FUNCTION_BLOCK "GCS7_E_MessageCtrl"	// FB 25
TITLE = MSG
//  
//COPYRIGHT:    (C) 1996 BY  BUHLER LTD.
//                           CH-9240 UZWIL  SWITZERLAND
//
//PRODUCT:      GCS7
//
//TITLE:        ELEMENT Control Message
//
//-------------------------------------------------------------------------
//
//IDENT:        AUTHOR:             DEPT:                       DATE:
//
//FB25.2.0      A. Egli             CT3                        17-Jun-2002
//              New Release with one block 
//FB25.1A       A.Egli              AEE61                      05-Feb-1997
//              1st Release in S7
//
//-------------------------------------------------------------------------
//
//PURPOSE:      MANUAL : see [MSGxxMAN]
//              Can send up to 16 diverent message to host
//
//RESTRICTIONS: S7
//              ACCU2: Pointer to dynamic datas of the element
//              ACCU1: Pointer to parameter datas of the element
//
//-------------------------------------------------------------------------
//
//=======================================================
//Log Message: 
//------------------------------------------------------
//0    Inp0           
//1    Inp1         
//     :  
//     :  
//14   Inp14      
//15   Inp15      
//
//=======================================================
//StCode:  State               
//------------------------------------------------------
//0    Inp0           
//1    Inp1         
//     :  
//     :  
//14   Inp14      
//15   Inp15      
//16   OK     
//
//
AUTHOR : EA
FAMILY : GCS7LL
NAME : MSG
VERSION : 2.0
VAR
  StCode : INT ;	//Element state code
  InMsg0 : BOOL ;	//Send Message 0
  InMsg1 : BOOL ;	//Send Message 1
  InMsg2 : BOOL ;	//Send Message 2
  InMsg3 : BOOL ;	//Send Message 3
  InMsg4 : BOOL ;	//Send Message 4
  InMsg5 : BOOL ;	//Send Message 5
  InMsg6 : BOOL ;	//Send Message 6
  InMsg7 : BOOL ;	//Send Message 7
  InMsg8 : BOOL ;	//Send Message 8
  InMsg9 : BOOL ;	//Send Message 9
  InMsg10 : BOOL ;	//Send Message 10
  InMsg11 : BOOL ;	//Send Message 11
  InMsg12 : BOOL ;	//Send Message 12
  InMsg13 : BOOL ;	//Send Message 13
  InMsg14 : BOOL ;	//Send Message 14
  InMsg15 : BOOL ;	//Send Message 15
  OutFlag0 : BOOL ;	//Message 0 done
  OutFlag1 : BOOL ;	//Message 1 done
  OutFlag2 : BOOL ;	//Message 2 done
  OutFlag3 : BOOL ;	//Message 3 done
  OutFlag4 : BOOL ;	//Message 4 done
  OutFlag5 : BOOL ;	//Message 5 done
  OutFlag6 : BOOL ;	//Message 6 done
  OutFlag7 : BOOL ;	//Message 7 done
  OutFlag8 : BOOL ;	//Message 8 done
  OutFlag9 : BOOL ;	//Message 9 done
  OutFlag10 : BOOL ;	//Message 10 done
  OutFlag11 : BOOL ;	//Message 11 done
  OutFlag12 : BOOL ;	//Message 12 done
  OutFlag13 : BOOL ;	//Message 13 done
  OutFlag14 : BOOL ;	//Message 14 done
  OutFlag15 : BOOL ;	//Message 15 done
  Par : STRUCT
   ParObjectNo : INT ;	//Is used for communication with PC, e.g. for message
   ParMsgType : INT ;	//Is used for message (translation of state)
   ParHornCode : INT ;	//Is used by horn module
   ParDisable : STRUCT 	//Disable Message
    Msg0 : BOOL ;
    Msg1 : BOOL ;
    Msg2 : BOOL ;
    Msg3 : BOOL ;
    Msg4 : BOOL ;
    Msg5 : BOOL ;
    Msg6 : BOOL ;
    Msg7 : BOOL ;
    Msg8 : BOOL ;
    Msg9 : BOOL ;
    Msg10 : BOOL ;
    Msg11 : BOOL ;
    Msg12 : BOOL ;
    Msg13 : BOOL ;
    Msg14 : BOOL ;
    Msg15 : BOOL ;
   END_STRUCT ;
   ParHornOff : STRUCT 	//Disable Horn
    Msg0 : BOOL ;
    Msg1 : BOOL ;
    Msg2 : BOOL ;
    Msg3 : BOOL ;
    Msg4 : BOOL ;
    Msg5 : BOOL ;
    Msg6 : BOOL ;
    Msg7 : BOOL ;
    Msg8 : BOOL ;
    Msg9 : BOOL ;
    Msg10 : BOOL ;
    Msg11 : BOOL ;
    Msg12 : BOOL ;
    Msg13 : BOOL ;
    Msg14 : BOOL ;
    Msg15 : BOOL ;
   END_STRUCT ;
  END_STRUCT ;
END_VAR
VAR_TEMP
  tmpLOGvalue : WORD ;	//LOG value
  tmpReport : BOOL ;	//Global LOG all
  tmpOffsetInstanzDB : DINT ;
  tmpLenDyn : DINT ;
  tmpCntBit : DINT ;
  tmpAddrDynLoop : DINT ;
  tmpAddrParDisable : DINT ;
END_VAR
BEGIN
NETWORK
TITLE =  Start Global
      L     16;
      T     #tmpLenDyn;	//--> Len dynamic data in byte
      TAR2;
      L     DW#16#FFFFFF;
      AD;
      L     P##Par;
      +D;
      L     P#6.0;	//P##ParDisable
      +D;
      T     #tmpAddrParDisable;
NETWORK
TITLE = PC Control
//=== Test Object number =====================
      L     "SYS_DirectCtrlDB".PC.ObjectNo;	//PCControl.ObjectNo
      L     #Par.ParObjectNo;	//Input ObjectNo
      <>I;
      JC    Ctrl;
//=== Test OType      ========================
      L     1025;	//Input object type
      L     "SYS_DirectCtrlDB".PC.ObjectType;	//PCControl.ObjectType
      <>I;
      JC    Ctrl;
//=== Test Handshake =========================
      A     "SYS_DirectCtrlDB".PC.Hsk.FExamine;	// Handshake.FExamine
      JC    pExa;
      L     2;	// FcInit
      UC    "SYS_DirectCtrl";
      JU    Ctrl;
// Write parameter 
// Write new commands from PC to Interface of group 
// Examine
pExa: TAR2;	// Address Dynamic datas
      T     "SYS_DirectCtrlDB".GC.InDynAddr;	// -->PCControl.GC.InDynAddr
      L     #tmpLenDyn;	// Length Dynamic datas
      T     "SYS_DirectCtrlDB".GC.InDynLen;	// -->PCControl.GC.InDynLen
      L     0;
      T     "SYS_DirectCtrlDB".GC.InParaAddr;	// -->PCControl.GC.InParaAddr
      T     "SYS_DirectCtrlDB".GC.InParaLen;	// -->PCControl.GC.InParaLen
      L     1;	// Code FcExamine
      UC    "SYS_DirectCtrl";
      L     10;	//Revision
      T     "SYS_DirectCtrlDB".GC.Revision;
NETWORK
TITLE = AllState
NETWORK
TITLE = Log
//Message Type: 0 to 15 
//O = InMsg0
//15= InMsg15
// 
// Init Flag msg done (OutFlagXx) if InMsgXx=0
Ctrl: L     DIW [AR2,P#2.0];	// Load  Bit pattern InMsg0 ...InMsg15
      L     DIW [AR2,P#4.0];	// Load  Bit pattern OutFlag0 ...OutFlag15
      AW;
      T     DIW [AR2,P#4.0];	// Reset Bits pattern OutFlag0 ...OutFlag15
// 
// Test new Message to send;
      TAR2  #tmpAddrDynLoop;
      L     16;
NEX1: T     #tmpCntBit;
      LAR1  #tmpAddrParDisable;
      AN    DIX [AR1,P#0.0];	// ParDisable.MsgXx
      LAR1  #tmpAddrDynLoop;
      A     DIX [AR1,P#2.0];	// InMsgXx
      AN    DIX [AR1,P#4.0];	// OutFlagXx
      S     DIX [AR1,P#4.0];	// OutFlagXx
      JC    LOG;
      +AR1  P#0.1;
      TAR1  #tmpAddrDynLoop;
      L     #tmpAddrParDisable;
      L     P#0.1;
      +D;
      T     #tmpAddrParDisable;
      L     #tmpCntBit;
      LOOP  NEX1;
      JU    OUT;
LOG:  L     B#(4, 16);	//MessageClass Info ""Message 16"
      L     #tmpCntBit;
      -I;
      T     #tmpLOGvalue;
      LAR1  #tmpAddrParDisable;
      A     DIX [AR1,P#2.0];	// ParHornOff.MsgXx
      JC    Log3;
      CALL  "SYS_Horn_Code" (
           FcCode                   := 1,
           ParObjectType            := 1025,
           ParObjectNo              := #Par.ParObjectNo,
           ParHornCode              := #Par.ParHornCode);
Log3: CALL  "GCS7_LogConvert" (
           ObjectNo                 := #Par.ParObjectNo,
           MsgType                  := #Par.ParMsgType,
           ClassMsgTxt              := #tmpLOGvalue,
           OType                    := 1025);	// LOG Message Converter / Entry / Contains Class and TextNo
NETWORK
TITLE = State Code
OUT:  LAR1  AR2;
      L     16;
NEX2: T     #tmpCntBit;
      A     DIX [AR1,P#2.0];	// InMsgXx
      JC    STC;
      +AR1  P#0.1;
      L     #tmpCntBit;
      LOOP  NEX2;
      L     16;
      JU    OK;
STC:  L     16;
      L     #tmpCntBit;
      -I;	// Code: fault
OK:   L     #StCode;	// Old state code
      TAK;
      T     #StCode;	// Save state code
      <>I;
      L     3;	// Load code for CBit methode
      CC    "SYS_CBitCtrl";
END_FUNCTION_BLOCK

FUNCTION_BLOCK "GCS7_E_DFCO"	// FB 26
TITLE = DFCO
//  
//COPYRIGHT:    (C) 1996  BUHLER AG, CH-9240 UZWIL, SWITZERLAND
//
//PRODUCT:      GCS7
//
//TITLE:        Element Control DFCO
//              (GCPROVB Revision 11)  
//
//-------------------------------------------------------------------------
//
//IDENT:        AUTHOR:             DEPT:                       DATE:
//
//FB26.2.3      A. Egli             BASE                        20-Okt-2008
//              For timeout starting check ParDFCO_Only
//FB26.2.2      A.Egli              CT3                         26-Sep-2007
//              Do not set "GCS7_Gr_InHeavyStartup" if ParDFCO_Only=1         
//FB26.2.1      A.Egli              CT3                         11-Sep-2007
//              Send Log Message if Alarmnumber changes from 0->X          
//FB26.2.0      A.Egli              CT3                         14-Feb-2007
//              New Tag names           
//FB26.1.4      B.Thoma             FU591                       02-Dez-2006
//              Delete all actual values as long Profibus fault           
//FB26.1.3      B.Thoma             FU91                        28-Nov-2006
//              Invert HL DFAV ; StCode Fan           
//FB26.1.2      B.Thoma             FU92                        18-Apr-2006
//              Flapbox changed 
//              FeedRoll State changed            
//FB26.1.1      A.Egli              CT3                         01-Dec-2005
//              Parameter Upload Change DBD86-->DBD88
//FB26.1.0      A.Egli              CT3                         06-Oct-2005
//              1st Release in S7
//
//-------------------------------------------------------------------------
//
//PURPOSE:      MANUAL : see [DFCOxxMAN]
//
//RESTRICTIONS: S7
//             
//=======================================================
//Log Message: 
//------------------------------------------------------
//0     = Fault Cancelled
//1..89 = AlarmLC : Alarmnumber see manual of MEAF
//90    = Fault Remote Control
//91    = StStopped
//92    = StStarted
//95    = WrongValue
//96    = Communication fault
//97    = 
//98    = 
//99    = Collected alarm
//
//=======================================================
//StCode:  State               
//------------------------------------------------------
// StFault                 32
// StStopped                1
// StStarting               2
// StStarted.Wait           3
// StStarted.Feeding        4
// StStopping               7
// StWarning                8
//
AUTHOR : EA
FAMILY : GCS7LL
NAME : DFCO
VERSION : 2.3
VAR
  StCode : INT ;	// State as code 32=StFault 1=StStopped 2=StStarting 3=StStartedWait 4=StStartedF
  spare20 : BOOL ;
  spare21 : BOOL ;
  spare22 : BOOL ;
  InReqStartRev : BOOL ;	//Mill must start reverse
  InReqStartFwd : BOOL ;	//Mill must start forward
  spare25 : BOOL ;	//1=Activate automatic control mode (CTRL.MODE)
  InHeavyFractionOpen : BOOL ;
  spare27 : BOOL ;
  spare30 : BOOL ;
  spare31 : BOOL ;	//
  CmdNext : BOOL ;	// Pulse to start the next motor in automatic mode
  CmdFaultReset : BOOL ;	// Command to reset fault
  InLocal : BOOL ;	// Local mode, accept all faults
  InManual : BOOL ;	//
  InReport : BOOL ;	//
  spare37 : BOOL ;
  InHWStop : BOOL ;	//HW stop is detected, no fault
  InDPFault : BOOL ;	//DP-Fault is detected, no fault
  InSimulation : BOOL ;	//Simulation with DPSim
  OutComFault : BOOL ;	//Communication fault
  OutStartwarning : BOOL ;	//Not used
  spare45 : BOOL ;
  spare46 : BOOL ;
  spare47 : BOOL ;
  StStopped : BOOL ;	//All motors are stopped
  StStarting : BOOL ;	//Not all relevant motors are started
  StStarted : BOOL ;	//All used motors are started
  StStopping : BOOL ;	//Any motor is stopping
  StFault : BOOL ;	//Any relevant element has a fault
  spare0505 : BOOL ;	//
  spare0506 : BOOL ;	//
  spare0507 : BOOL ;	//
  Mill1 : STRUCT
   InEnable : BOOL ;	//Automatic Mode
   InUsed : BOOL ;	//Automatic Mode
   InEnableFeed : BOOL ;	//Automatic Mode
   InBrake : BOOL ;	//Automatic Mode: Stop with break
   InFast : BOOL ;	//Run motor with fast speed
   spare05 : BOOL ;
   spare06 : BOOL ;
   spare07 : BOOL ;
   CmdOff : BOOL ;	//Manual Mode
   CmdOn : BOOL ;	//Manual Mode
   CmdFeedOff : BOOL ;	//Manual Mode
   CmdFeedOn : BOOL ;	//Manual Mode
   CmdBrake : BOOL ;	//Manual Mode
   spare15 : BOOL ;
   spare16 : BOOL ;
   InpFanStart : BOOL ;	//Fan is started
   OutpMotorFwd : BOOL ;	//Output run motor forward
   OutpMotorFast : BOOL ;	//Output run motor fast
   OutpMotorRev : BOOL ;	//Output run motor reverse
   OutpBrake : BOOL ;	//Output brake
   OutpFanStart : BOOL ;	//Output run fan
   OutLoaded : BOOL ;	//Read from DFCO
   OutWrongValue : BOOL ;
   OutScreenChangeReq : BOOL ;	//Srceen change is requested
   VarEdgeStarted : BOOL ;
   VarEdgeFault : BOOL ;
   Tar : STRUCT 	//Telegram Dataset 128
    InSetPoint : INT ;	//[%] Load control
    InScreen : INT ;	//[0.1mm] Sreen size
    spare1 : INT ;
    spare2 : INT ;
    spare3 : INT ;
    spare4 : INT ;
    EmptyTime : INT ;	//[0.1s]
    spare5 : INT ;
   END_STRUCT ;
   Act : STRUCT 	//Telegram Dataset 1
    OutLoadAct : INT ;	//[%]
    OutCurrentLoad : INT ;	//[0.1A]
    OutActPosSlide : INT ;	//[%]
    OutActTemperature : INT ;	//[0.1°C]
    OutStatusFlapBox : INT ;
    OutStatusMillMotor : INT ;
    spare1 : INT ;
    OutEmptyTime : INT ;	//[0.1s]
    spare2 : INT ;
    OutAlarmNo : INT ;
   END_STRUCT ;
   Motor : STRUCT
    StStopped : BOOL ;
    StStarting : BOOL ;
    StStartedFwd : BOOL ;
    StStopping : BOOL ;
    StFault : BOOL ;
    StStartedRev : BOOL ;
    StBrake : BOOL ;
   END_STRUCT ;
   OutScreenAct : INT ;	//[0.1mm] Actual screen
   spare1 : INT ;
   spare2 : INT ;
   spare3 : INT ;
   spare4 : INT ;
   spare5 : INT ;
   spare6 : INT ;
   Motor_StCode : INT ;	//StCode same as EL_Motor
   Vibration_StCode : INT ;	//StCode same as EL_DIC
   Automatic_StCode : INT ;	//StCode same as EL_DIC
   StandStill_StCode : INT ;	//StCode same as EL_DIC
   SwitchPanel_StCode : INT ;	//StCode same as EL_DIC
   EmergencyStop_StCode : INT ;	//StCode same as EL_DIC
   HLCone_StCode : INT ;	//StCode same as EL_DIC
   OutTimeStartedFwd : DINT ;	//[s] Not errasable time "Started"
   OutTimeStartedRev : DINT ;	//[s] Not errasable time "Started"
   OutTimeFaulted : DINT ;	//[s] Not errasable time "Faulted"
   OutCntStartup : DINT ;	//Not errasable counter of startup
   OutCntFault : DINT ;	//Not errasable counter of faults
  END_STRUCT ;
  Mill2 : STRUCT
   InEnable : BOOL ;	//Automatic Mode
   InUsed : BOOL ;	//Automatic Mode
   InEnableFeed : BOOL ;	//Automatic Mode
   InBrake : BOOL ;	//Automatic Mode: Stop with break
   InFast : BOOL ;	//Run motor with fast speed
   spare05 : BOOL ;
   spare06 : BOOL ;
   spare07 : BOOL ;
   CmdOff : BOOL ;	//Manual Mode
   CmdOn : BOOL ;	//Manual Mode
   CmdFeedOff : BOOL ;	//Manual Mode
   CmdFeedOn : BOOL ;	//Manual Mode
   CmdBrake : BOOL ;	//Manual Mode
   spare15 : BOOL ;
   spare16 : BOOL ;
   InpFanStart : BOOL ;	//Fan is started
   OutpMotorFwd : BOOL ;	//Output run motor forward
   OutpMotorFast : BOOL ;	//Output run motor fast
   OutpMotorRev : BOOL ;	//Output run motor reverse
   OutpBrake : BOOL ;	//Output brake
   OutpFanStart : BOOL ;	//Output run fan
   OutLoaded : BOOL ;	//Read from DFCO
   OutWrongValue : BOOL ;
   OutScreenChangeReq : BOOL ;	//Srceen change is requested
   VarEdgeStarted : BOOL ;
   VarEdgeFault : BOOL ;
   Tar : STRUCT 	//Telegram Dataset 128
    InSetPoint : INT ;	//[%] Load control
    InScreen : INT ;	//[0.1mm] Sreen size
    spare1 : INT ;
    spare2 : INT ;
    spare3 : INT ;
    spare4 : INT ;
    EmptyTime : INT ;	//[0.1s]
    spare5 : INT ;
   END_STRUCT ;
   Act : STRUCT 	//Telegram Dataset 1
    OutLoadAct : INT ;	//[%]
    OutCurrentLoad : INT ;	//[0.1A]
    OutActPosSlide : INT ;	//[%]
    OutActTemperature : INT ;	//[0.1°C]
    OutStatusFlapBox : INT ;
    OutStatusMillMotor : INT ;
    spare1 : INT ;
    OutEmptyTime : INT ;	//[0.1s]
    spare2 : INT ;
    OutAlarmNo : INT ;
   END_STRUCT ;
   Motor : STRUCT
    StStopped : BOOL ;
    StStarting : BOOL ;
    StStartedFwd : BOOL ;
    StStopping : BOOL ;
    StFault : BOOL ;
    StStartedRev : BOOL ;
    StBrake : BOOL ;
   END_STRUCT ;
   OutScreenAct : INT ;	//[0.1mm] Actual screen
   spare1 : INT ;
   spare2 : INT ;
   spare3 : INT ;
   spare4 : INT ;
   spare5 : INT ;
   spare6 : INT ;
   Motor_StCode : INT ;	//StCode same as EL_Motor
   Vibration_StCode : INT ;	//StCode same as EL_DIC
   Automatic_StCode : INT ;	//StCode same as EL_DIC
   StandStill_StCode : INT ;	//StCode same as EL_DIC
   SwitchPanel_StCode : INT ;	//StCode same as EL_DIC
   EmergencyStop_StCode : INT ;	//StCode same as EL_DIC
   HLCone_StCode : INT ;	//StCode same as EL_DIC
   OutTimeStartedFwd : DINT ;	//[s] Not errasable time "Started"
   OutTimeStartedRev : DINT ;	//[s] Not errasable time "Started"
   OutTimeFaulted : DINT ;	//[s] Not errasable time "Faulted"
   OutCntStartup : DINT ;	//Not errasable counter of startup
   OutCntFault : DINT ;	//Not errasable counter of faults
  END_STRUCT ;
  OutActFeedRoll : INT ;	//[Hz] Actual frequence feed roll
  spare208 : DINT ;	//StCode same as EL_DIC
  spare212 : DINT ;
  spare216 : DINT ;
  FlapBox : STRUCT
   StMill1 : BOOL ;
   StMiddle : BOOL ;
   StMill2 : BOOL ;
   StNoPosition : BOOL ;
  END_STRUCT ;
  FlapBox_StCode : INT ;	//StCode same as EL_VLS4
  FeedRoll_StCode : INT ;	//StCode same as EL_Motor
  Fan_StCode : INT ;	//StCode same as EL_Motor
  LL_FeedHopper_StCode : INT ;	//StCode same as EL_DIC
  HL_DFAV_StCode : INT ;	//StCode same as EL_DIC
  MagnetDoor_StCode : INT ;	//StCode same as EL_DIC
  HeavyParticalFlap_StCode : INT ;	//StCode same as EL_DIC
  spare118 : INT ;
  spare220 : DINT ;
  spare224 : DINT ;
  spare228 : DINT ;
  OutAlarmNoLog : INT ;	//Last textnumber send to log
  InpDFCO : STRUCT 	//WAGO/MEAF Inputs of DFCO
   I00_LL_FeedHopper : BOOL ;	//DFAV: Inlet level DFAV (1=covered)
   I01_HL_DFAV : BOOL ;	//DFAV: High level DFAV (1=Covered)
   I02_HeavyParticleFlap : BOOL ;	//DFAV: Heavy particle flap closed (1=end position)
   I03_MagnetDoorClosed : BOOL ;	//DFAV: Door interlocking heavy particle flap (1=closed)
   I04_LSFlapBox : BOOL ;	//DFAV: LS of middle position (1=dedected)
   I05 : BOOL ;
   I06 : BOOL ;
   I07_24VOk : BOOL ;	//DFAV: Fuse control of DFCO (1=ok)
   spare9 : BYTE ;
   I20_ButtonCone1 : BOOL ;	//DFZK Mill 1: Button open/close cone
   I21_ButtonHeavyFlap1 : BOOL ;	//DFZK Mill 1: Button open heavy particle flap
   I22_KeySwitchAuto1 : BOOL ;	//DFZK Mill 1: Key switch Automatic/Hand (1=Hand)
   I23_SwitchPanel1 : BOOL ;	//DFZK Mill 1: Connection box (1= inactive)
   I24_StandStill1 : BOOL ;	//DFZK Mill 1: Standstill (1=Standstill)
   I25_EmergencyStop1 : BOOL ;	//DFZK Mill 1: Cone interlocking (1=not interlocked)
   I26_EmergencySwitch1 : BOOL ;	//DFZK Mill 1: Emergency switch(1=ok)
   I27_HL_Cone1 : BOOL ;	//DFZK Mill 1: HL outlet cone (1=uncovered)
   spare11 : BYTE ;
   I40_ButtonCone2 : BOOL ;	//DFZK Mill 2: Button open/close cone
   I41_ButtonHeavyFlap2 : BOOL ;	//DFZK Mill 2: Button open heavy particle flap
   I42_KeySwitchAuto2 : BOOL ;	//DFZK Mill 2: Key switch Automatic/Hand (1=Hand)
   I43_SwitchPanel2 : BOOL ;	//DFZK Mill 2: Connection box (1= inactive)
   I44_StandStill2 : BOOL ;	//DFZK Mill 2: Standstill (1=Standstill)
   I45_EmergencyStop2 : BOOL ;	//DFZK Mill 2: Cone interlocking (1=not interlocked)
   I46_EmergencySwitch2 : BOOL ;	//DFZK Mill 2: Emergency switch(1=ok)
   I47_HL_Cone2 : BOOL ;	//DFZK Mill 2: HL outlet cone (1=uncovered)
   spare13 : BYTE ;
   I60_VibrationDetector1 : BOOL ;	//DFZK Mill 1: Vibration detector (1=OK)
   I61_VibrationDetector2 : BOOL ;	//DFZK Mill 2: Vibration detector (1=OK)
   spare15 : BYTE ;
   I80_Release1 : BOOL ;	//DFZK Mill 1: Release feeding (1=released)
   I81_Start1 : BOOL ;	//DFZK Mill 1: Release motor (1=released)
   I82_RotarySpeed1 : BOOL ;	//DFZK Mill 1: Fast/Slow speed of motor (2=fast)
   I83_AckFan : BOOL ;	//DFZK Mill 1: Fan is running
   I84 : BOOL ;
   I85 : BOOL ;
   I86 : BOOL ;
   I87 : BOOL ;
   I90_Release2 : BOOL ;	//DFZK Mill 2: Release feeding (1=released)
   I91_Start2 : BOOL ;	//DFZK Mill 2: Release motor (1=released)
   I92_Speed2 : BOOL ;	//DFZK Mill 2: Fast/Slow speed of motor (1=fast)
   I93_Break : BOOL ;	//DFZK Mill 1/2: Stop with break (1=with break)
   spare18 : BYTE ;
   spare19 : BYTE ;
   spare20 : BYTE ;
   DI1_spare : BOOL ;
   DI2_spare : BOOL ;
   DI3_spare : BOOL ;
   DI4_spare : BOOL ;
   DI5_SlideEndPos1 : BOOL ;	//DFZK Mill 1: Slide end position
   DI6_SlidePulse1 : BOOL ;	//DFZK Mill 1: Slide pulse signal
   DI7_SlideEndPos2 : BOOL ;	//DFZK Mill 2: Slide end position
   DI8_SlidePulse2 : BOOL ;	//DFZK Mill 2: Slide pulse signal
  END_STRUCT ;
  OutpDFCO : STRUCT 	//WAGO/MEAF Outpus of DFCO
   O00_HeavyParticleClose : BOOL ;	//DFAV: Heavy particle flap close
   O01_HeavyParticleOpen : BOOL ;	//DFAV: Heavy particle flap open
   O02_FlapCylinderExtend : BOOL ;	//DFAV: Flap box cylinder extend
   O03_FlapCylinderRetract : BOOL ;	//DFAV: Flap box cylinder retract
   spare9 : BYTE ;
   O20_LampAlarm1 : BOOL ;	//DFZK Mill 1: Lamp alarm (1=Alarm)
   O21_LampRelaseCone1 : BOOL ;	//DFZK Mill 1: Lamp cone adjustment
   O22_LampHeavyParticle : BOOL ;	//DFZK Mill 1: Lamp heavy particle flap
   spare11 : BYTE ;
   O40_LampAlarm2 : BOOL ;	//DFZK Mill 2: Lamp alarm (1=Alarm)
   O41_LampReleaseCone2 : BOOL ;	//DFZK Mill 2: Lamp cone adjustment
   O42_LampHeavyParticle : BOOL ;	//DFZK Mill 2: Lamp heavy particle flap
   O43 : BOOL ;
   O44 : BOOL ;
   O45 : BOOL ;
   O46 : BOOL ;
   O47 : BOOL ;
   O50_ConeOpen1 : BOOL ;	//DFZK Mill 1: Cone open
   O51_ConeClose1 : BOOL ;	//DFZK Mill 1: Cone close
   O52 : BOOL ;	//
   O53 : BOOL ;	//
   O54 : BOOL ;
   O55 : BOOL ;
   O56 : BOOL ;
   O57 : BOOL ;
   O60_ConeOpen2 : BOOL ;	//DFZK Mill 2: Cone open
   O61_ConeClose2 : BOOL ;	//DFZK Mill 2: Cone close
   spare15 : BYTE ;
   O80_Alarm1 : BOOL ;	//DFZK Mill 1: Alarm (1=no alarm)
   O81_StartMotor1 : BOOL ;	//DFZK Mill 1: Start motor forward
   O82_MotorFast1 : BOOL ;	//DFZK Mill 1: Start motor fast
   O83_MotorRev1 : BOOL ;	//DFZK Mill 1: Start motor reverse
   O84_Break1 : BOOL ;	//DFZK Mill 1: Brake motor
   O85_StartFan : BOOL ;	//DFZK Mill 1/2: Start fan
   O86 : BOOL ;
   O87 : BOOL ;
   O90_Alarm2 : BOOL ;	//DFZK Mill 2: Alarm (1=no alarm)
   O91_StartMotor2 : BOOL ;	//DFZK Mill 2: Start motor forward
   O92_MotorFast2 : BOOL ;	//DFZK Mill 2: Start motor fast
   O93_MotorRev2 : BOOL ;	//DFZK Mill 2: Start motor reverse
   O94_Break2 : BOOL ;	//DFZK Mill 2: Brake motor
   spare18 : BYTE ;
   spare19 : BYTE ;
   spare20 : BYTE ;
   DO1_SummaryAlarm : BOOL ;	//Summary alarm
   DO2 : BOOL ;
   DO3 : BOOL ;
   DO4_Slide1Open : BOOL ;	//Slide 1 open
   DO5_Slide1Close : BOOL ;	//Slide 1 close
   DO6_Slide2Open : BOOL ;	//Slide 2 open
   DO7_Slide2Close : BOOL ;	//Slide 2 close
   DO8 : BOOL ;
  END_STRUCT ;
  Command : STRUCT 	//Command for DFCO
   spare0 : BOOL ;	//1=Automatic/ 0=Manual
   AckStartRequest : BOOL ;	//Acknowledge Start Request
   ReqStartRev : BOOL ;	//Mill must start reverse
   ReqStartFwd : BOOL ;	//Mill must start forward
   HeavyFractionOpen : BOOL ;	//Heavy fraction flap is open
   ReqScreenChange1 : BOOL ;
   ReqScreenChange2 : BOOL ;
   AcceptNewDataReady : BOOL ;	//de: Quittierung neue Werte Bereit
   EnableMill1 : BOOL ;	//Enable to start mill 1
   MotorMill1Fast : BOOL ;
   UsedMill1 : BOOL ;
   BrakeMill1 : BOOL ;	//Stop mill 1
   EnableFeedMill1 : BOOL ;	//Enable Feed of mill 1
   AckFanStart : BOOL ;	//Fan is running
   spare16 : BOOL ;
   spare17 : BOOL ;
   EnableMill2 : BOOL ;	//Enable to start mill 1
   MotorMill2Fast : BOOL ;
   UsedMil12 : BOOL ;
   BrakeMill2 : BOOL ;	//Stop mill 1
   EnableFeedMill2 : BOOL ;	//Enable Feed of mill 1
   spare25 : BOOL ;
   spare26 : BOOL ;
   spare27 : BOOL ;
   CommandReady : BOOL ;	//de: Steuersignale gültig
   spare41 : BOOL ;
   spare42 : BOOL ;
   spare43 : BOOL ;
   spare44 : BOOL ;
   ResetAlarm : BOOL ;	//de: Alarm löschen
   NewSendData : BOOL ;	//de: Aenderung Sendedaten
   AcceptNewRcvData : BOOL ;	//de: Quittierung Aenderung Empfangsdatensatz
  END_STRUCT ;
  Status : STRUCT 	//Status from DFCO
   spare00 : BOOL ;
   ReqStartRequest : BOOL ;	//Start Request : DFCO like to start a motor
   Loaded1 : BOOL ;	//Mill 1 loaded with product
   Loaded2 : BOOL ;	//Mill 2 loaded with product
   spare04 : BOOL ;
   AckScreenChange1 : BOOL ;
   AckScreenChange2 : BOOL ;
   NewDataReady : BOOL ;	//de: Neue Werte Bereit
   O80Alarm1 : BOOL ;	//False=Alarm
   O81MotorFwd1 : BOOL ;	//Output run motor forward
   O82MotorFast1 : BOOL ;	//Output run motor fast
   O83MotorRev1 : BOOL ;	//Output run motor reverse
   O84Brake1 : BOOL ;	//Output brake
   O85FanStart : BOOL ;	//Output run fan
   spare16 : BOOL ;
   spare17 : BOOL ;
   O90Alarm2 : BOOL ;	//False=Alarm
   O91MotorFwd2 : BOOL ;	//Output run motor forward
   O92MotorFast2 : BOOL ;	//Output run motor fast
   O93MotorRev2 : BOOL ;	//Output run motor reverse
   O94Brake2 : BOOL ;	//Output brake
   spare25 : BOOL ;	//Output run fan
   spare26 : BOOL ;
   spare27 : BOOL ;
   spare30 : BOOL ;
   spare31 : BOOL ;
   spare32 : BOOL ;	//de: Stuerung Remote
   RemoteControlDP : BOOL ;	//de: Sollwertvorgabe Remote
   WrongValue : BOOL ;	//de: Falscher Sollwert
   SumFault : BOOL ;	//de: Sammelalarm
   AcceptNewSendData : BOOL ;	//de: Quittierung Aenderung Sendedaten
   NewRcvData : BOOL ;	//de: Aenderung Empfangsdaten
  END_STRUCT ;
  Par : STRUCT
   ParObjectNo : INT ;	//Is used for communication with PC, e.g. for message
   ParMsgType : INT ;	//Is used for message (translation of state)
   ParHornCode : INT ;	//Is used by horn module
   ParLogOff : BOOL ;	//Report is off
   ParManual : BOOL ;	//Manual mode without interlocking
   ParDFCO_Only : BOOL ;	//Only throughput regulation, no motors
   ParStartwarning : BOOL ;	//not used
   ParIOByteNo : INT ;	//PROFIBUS: Address of first input and output byte Profibus DP
   ParTimeOutStart : INT  := 50;	//[0.1s] After this time the motor must start
   OutTimeOutStart1 : INT ;	//[0.1s] Actual timeout time mill 1
   OutTimeOutStart2 : INT ;	//[0.1s] Actual timeout time mill 2
   Spare94 : DINT ;
   spare98 : DINT ;
   Spare94_1 : DINT ;
   HelpFlags : STRUCT 	//Aux. signal to retry fault message
    OutFaultResetDone : BOOL ;
    OutTestNewAlarm : BOOL ;
    OutFlagFaultResetDone : BOOL ;
    OutComFaultRead : BOOL ;
    OutComFaultSend : BOOL ;
   END_STRUCT ;
  END_STRUCT ;
END_VAR
VAR_TEMP
  tmpLOGvalue : WORD ;	//LOG value
  tmpReport : BOOL ;	//Global LOG all
  tmpFault : BOOL ;
  tmpLocal : BOOL ;
  tmpStarted : BOOL ;
  tmpStopped : BOOL ;
  tmpLenDyn : DINT ;
  tmpReturn : INT ;
  DPData : STRUCT
   StatusCommand : DWORD ;
   NrSndDataSet : BYTE ;	//de: Nummer Sendedatensatz
   IdxSndDataSet : BYTE ;	//de: Index Sendedatensatz
   NrRcvDataSet : BYTE ;	//de: Nummer Empfangsdatensatz
   IdxRcvDataSet : BYTE ;	//de: Index Empfangsdatensatz
   Data : ARRAY  [1 .. 4 ] OF DINT ;
  END_STRUCT ;
  Set1 : STRUCT
   OutLoadAct : INT ;	//[%]
   OutCurrentLoad : INT ;	//[0.1A]
   OutActPosSlide : INT ;	//[%]
   OutActTemperature : INT ;	//[0.1°C]
   OutStatusFlapBox : BYTE ;
   OutStatusMillMotor : BYTE ;
   OutActFeedFoll : BYTE ;	//[Hz] Actual frequence feed roll
   spare1 : BYTE ;
   OutEmptyTime : INT ;	//[0.1s]
   spare2 : BYTE ;
   OutAlarmNo : BYTE ;
  END_STRUCT ;
  tmpAddr : WORD ;
  tmpCnt : INT ;
  tmpRetVal : INT ;
  tmpBool : BOOL ;
END_VAR
BEGIN
NETWORK
TITLE =  Start Global
      L     298;
      T     #tmpLenDyn;	//--> Len dynamic data in byte
NETWORK
TITLE = PC Control
//=== Test Object number =====================
      L     "SYS_DirectCtrlDB".PC.ObjectNo;	//PCControl.ObjectNo
      L     #Par.ParObjectNo;	//Input ObjectNo
      <>I;
      JC    aEnd;
//=== Test OType  ========================
      L     1026;	//Input object type
      L     "SYS_DirectCtrlDB".PC.ObjectType;	//PCControl.ObjectType
      <>I;
      JC    aEnd;
//=== Test Handshake =========================
      A     "SYS_DirectCtrlDB".PC.Hsk.FExamine;	// Handshake.FExamine
      JC    aExa;
      A     "SYS_DirectCtrlDB".PC.Hsk.FDefineCmd;	// Handshake.FDefineCmd
      JC    aCmd;
      A     "SYS_DirectCtrlDB".PC.Hsk.FDefinePara;	// Handshake.FDefinePara
      JC    pPar;
aIni: L     2;	// FcInit
      UC    "SYS_DirectCtrl";
      JU    aEnd;
// Write parameter 
pPar: LAR1  P#DBX 58.0;
      L     P#6.0;
      +AR1;
// Write new commands from PC to Interface of group 
// Mill 1
aCmd: A     "SYS_DirectCtrlDB".PC.Cmd1[0];	//CmdBrakeMill1On
      AN    "GCS7_Gr_OutManualOff";	//Global.OutManualOff  [2.10]
      S     #Mill1.CmdBrake;
      A     "SYS_DirectCtrlDB".PC.Cmd1[1];	//CmdReqSlow
      R     #Command.MotorMill1Fast;
      A     "SYS_DirectCtrlDB".PC.Cmd1[2];	//CmdReqFast
      S     #Command.MotorMill1Fast;
      A     "SYS_DirectCtrlDB".PC.Cmd1[3];	//CmdReqRev
      S     #Command.ReqStartRev;
      R     #Command.ReqStartFwd;
      A     "SYS_DirectCtrlDB".PC.Cmd1[4];	//CmdReqFwd
      R     #Command.ReqStartRev;
      S     #Command.ReqStartFwd;
      A     "SYS_DirectCtrlDB".PC.Cmd1[8];	// CmdOff
      AN    "GCS7_Gr_OutManualOff";	//Global.OutManualOff  [2.10]
      S     #Mill1.CmdOff;
      A     "SYS_DirectCtrlDB".PC.Cmd1[9];	// CmdOn
      AN    "GCS7_Gr_OutManualOff";	//Global.OutManualOff  [2.10]
      S     #Mill1.CmdOn;
      A     "SYS_DirectCtrlDB".PC.Cmd1[6];	// CmdFeedOff
      AN    "GCS7_Gr_OutManualOff";	//Global.OutManualOff  [2.10]
      S     #Mill1.CmdFeedOff;
      A     "SYS_DirectCtrlDB".PC.Cmd1[7];	// CmdFeedOn
      AN    "GCS7_Gr_OutManualOff";	//Global.OutManualOff  [2.10]
      S     #Mill1.CmdFeedOn;
// Mill 2
      A     "SYS_DirectCtrlDB".PC.Cmd2[0];	//Cmd1[0]=CmdBrakeMill1On
      AN    "GCS7_Gr_OutManualOff";	//Global.OutManualOff  [2.10]
      S     #Mill2.CmdBrake;
      A     "SYS_DirectCtrlDB".PC.Cmd2[1];	//CmdReqSlow
      R     #Command.MotorMill2Fast;
      A     "SYS_DirectCtrlDB".PC.Cmd2[2];	//CmdReqFast
      S     #Command.MotorMill2Fast;
      A     "SYS_DirectCtrlDB".PC.Cmd2[8];	// CmdOff
      AN    "GCS7_Gr_OutManualOff";	//Global.OutManualOff  [2.10]
      S     #Mill2.CmdOff;
      A     "SYS_DirectCtrlDB".PC.Cmd2[9];	// CmdOn
      AN    "GCS7_Gr_OutManualOff";	//Global.OutManualOff  [2.10]
      S     #Mill2.CmdOn;
      A     "SYS_DirectCtrlDB".PC.Cmd2[6];	// CmdFeedOff
      AN    "GCS7_Gr_OutManualOff";	//Global.OutManualOff  [2.10]
      S     #Mill2.CmdFeedOff;
      A     "SYS_DirectCtrlDB".PC.Cmd2[7];	// CmdFeedOn
      AN    "GCS7_Gr_OutManualOff";	//Global.OutManualOff  [2.10]
      S     #Mill2.CmdFeedOn;
// Mill 1+2
//-> [1.3] Tho: tlw. geändert; Reihenfolge korrig.
      A     "SYS_DirectCtrlDB".PC.Cmd1[10];	// CmdNext
      S     #CmdNext;
      A     "SYS_DirectCtrlDB".PC.Cmd1[11];	// CmdFaultReset
      S     #CmdFaultReset;
      A     "SYS_DirectCtrlDB".PC.Cmd1[13];	// CmdManualOn
      S     #InManual;
      A     "SYS_DirectCtrlDB".PC.Cmd2[13];	// CmdManualOff
      R     #InManual;
      A     "SYS_DirectCtrlDB".PC.Cmd1[14];	// CmdReportOn
      S     #InReport;
      A     "SYS_DirectCtrlDB".PC.Cmd2[14];	// CmdReportOff
      R     #InReport;
//<- [1.3]
      JU    aIni;
aExa: TAR2;	// Address Dynamic datas
      T     "SYS_DirectCtrlDB".GC.InDynAddr;	// -->PCControl.GC.InDynAddr
      L     #tmpLenDyn;	// Length Dynamic data
      T     "SYS_DirectCtrlDB".GC.InDynLen;	// -->PCControl.GC.InDynLen
      L     0;
      T     "SYS_DirectCtrlDB".GC.InParaAddr;	// -->PCControl.GC.InParaAddr
      T     "SYS_DirectCtrlDB".GC.InParaLen;	// -->PCControl.GC.InParaLen
      L     1;	// Code FcExamine
      UC    "SYS_DirectCtrl";
      L     11;	//Revision
      T     "SYS_DirectCtrlDB".GC.Revision;
aEnd: NOP   0;
NETWORK
TITLE = (Profibus) Read data
      L     #Par.ParIOByteNo;
      T     #tmpAddr;
      A     #InSimulation;
      JC    rSim;
      CALL  "SIEMENS_DPRD_DAT" (
           LADDR                    := #tmpAddr,
           RET_VAL                  := #tmpReturn,
           RECORD                   := #DPData);
      L     #tmpReturn;
      L     0;
      <>I;
      =     #Par.HelpFlags.OutComFaultRead;
      JC    rcv0;
      JU    rDP;
//read from Simulation
rSim: R     #Par.HelpFlags.OutComFaultRead;
      A     "GCS7_Gr_SimDPtoImage";
      L     P#I 0.0;
      JC    rDB1;
      OPN   "TEST_IOSimuliInput";
      L     P#DBX 0.0;
rDB1: L     #Par.ParIOByteNo;
      SLD   3;
      +D;
      LAR1;
      L     D [AR1,P#0.0];
      T     #DPData.StatusCommand;
      L     B [AR1,P#4.0];
      T     #DPData.NrSndDataSet;
      L     B [AR1,P#5.0];
      T     #DPData.IdxSndDataSet;
      L     B [AR1,P#6.0];
      T     #DPData.NrRcvDataSet;
      L     B [AR1,P#7.0];
      T     #DPData.IdxRcvDataSet;
      L     D [AR1,P#8.0];
      T     #DPData.Data[1];
      L     D [AR1,P#12.0];
      T     #DPData.Data[2];
      L     D [AR1,P#16.0];
      T     #DPData.Data[3];
      L     D [AR1,P#20.0];
      T     #DPData.Data[4];
//==Copy Status===============
rDP:  L     #DPData.NrRcvDataSet;
      L     0;
      ==I;
      JC    R101;
      CALL  "SIEMENS_BLKMOV" (
           SRCBLK                   := #DPData.StatusCommand,
           RET_VAL                  := #tmpReturn,
           DSTBLK                   := #Status);
      AN    #Status.NewRcvData;
      A     #InSimulation;
      JC    rcv0;
      CALL  "SIEMENS_BLKMOV" (
           SRCBLK                   := #DPData.Data,
           RET_VAL                  := #tmpReturn,
           DSTBLK                   := #Set1);
//===============================
//Answer Dataset 001 Index 1
      L     #DPData.NrRcvDataSet;
      L     1;
      <>I;
      O;
      O(;
      L     #DPData.IdxRcvDataSet;
      L     1;
      <>I;
      );
      JC    r201;
      L     #Set1.OutLoadAct;
      T     #Mill1.Act.OutLoadAct;
      L     #Set1.OutActFeedFoll;
      T     #OutActFeedRoll;
      L     #Set1.OutCurrentLoad;
      T     #Mill1.Act.OutCurrentLoad;
      L     #Set1.OutActPosSlide;
      T     #Mill1.Act.OutActPosSlide;
      L     #Set1.OutActTemperature;
      T     #Mill1.Act.OutActTemperature;
      L     #Set1.OutStatusFlapBox;
      T     #Mill1.Act.OutStatusFlapBox;
      L     #Set1.OutStatusMillMotor;
      T     #Mill1.Act.OutStatusMillMotor;
      L     #Set1.spare1;
      T     #Mill1.Act.spare1;
      L     #Set1.OutEmptyTime;
      T     #Mill1.Act.OutEmptyTime;
      L     #Set1.spare2;
      T     #Mill1.Act.spare2;
      L     #Set1.OutAlarmNo;
      T     #Mill1.Act.OutAlarmNo;
      JU    R201;	//[7.0]   
//===============================
//Answer Dataset 1 Index 2
r201: L     #DPData.NrRcvDataSet;
      L     1;
      <>I;
      O;
      O(;
      L     #DPData.IdxRcvDataSet;
      L     2;
      <>I;
      );
      JC    r002;
      L     #Set1.OutLoadAct;
      T     #Mill2.Act.OutLoadAct;
      L     #Set1.OutActFeedFoll;
      T     #OutActFeedRoll;
      L     #Set1.OutCurrentLoad;
      T     #Mill2.Act.OutCurrentLoad;
      L     #Set1.OutActPosSlide;
      T     #Mill2.Act.OutActPosSlide;
      L     #Set1.OutActTemperature;
      T     #Mill2.Act.OutActTemperature;
      L     #Set1.OutStatusFlapBox;
      T     #Mill2.Act.OutStatusFlapBox;
      L     #Set1.OutStatusMillMotor;
      T     #Mill2.Act.OutStatusMillMotor;
      L     #Set1.spare1;
      T     #Mill2.Act.spare1;
      L     #Set1.OutEmptyTime;
      T     #Mill2.Act.OutEmptyTime;
      L     #Set1.spare2;
      T     #Mill2.Act.spare2;
      L     #Set1.OutAlarmNo;
      T     #Mill2.Act.OutAlarmNo;
      JU    R002;
//Answer  dataset 2  : Wago/MEAF Inputs
r002: L     #DPData.NrRcvDataSet;
      L     2;
      <>I;
      JC    r003;
      CALL  "SIEMENS_BLKMOV" (
           SRCBLK                   := #DPData.Data,
           RET_VAL                  := #tmpReturn,
           DSTBLK                   := #InpDFCO);
      JU    R003;
//Answer  dataset 3  : Wago/MEAF Outputs
r003: L     #DPData.NrRcvDataSet;
      L     3;
      <>I;
      JC    r011;
      CALL  "SIEMENS_BLKMOV" (
           SRCBLK                   := #DPData.Data,
           RET_VAL                  := #tmpReturn,
           DSTBLK                   := #OutpDFCO);
      JU    R011;
//---Answer  dataset 11 ---
//---Answer  dataset 12 ---
r011: L     #DPData.NrRcvDataSet;
      L     11;
      <>I;
      JC    rLCB;
// Answer Dataset 11
      L     '  ';
      T     "SYS_DirectCtrlLCDB".PC.Value[1];
      L     #DPData.Data[1];
      T     DB10.DBD 60;
      L     #DPData.Data[2];
      T     DB10.DBD 64;
      L     #DPData.Data[3];
      T     DB10.DBD 68;
      L     #DPData.Data[4];
      T     DB10.DBD 72;
      L     #DPData.IdxRcvDataSet;
      L     255;
      ==I;
      JC    rLCE;
      S     "SYS_DirectCtrlLCDB".GC.Set11Done;
      L     12;
      T     #DPData.NrRcvDataSet;
      L     0;
      T     #DPData.IdxRcvDataSet;
      JU    rcv0;	//--> Read dataset 12
// Answer Dataset 12
rLCB: L     #DPData.NrRcvDataSet;
      L     12;
      <>I;
      JC    R101;
      L     #DPData.Data[1];
      T     DB10.DBD 76;
      L     #DPData.Data[2];
      T     DB10.DBD 80;
      L     #DPData.Data[3];
      T     DB10.DBD 84;
      L     #DPData.Data[4];
      T     DB10.DBD 88;
      AN    "SYS_DirectCtrlLCDB".GC.Set11Done;
      JC    R101;
rLCE: L     12;
      CALL  "SYS_DirectCtrl";
      JU    R101;
//===============================
//[7.0]--> LC Parameter 
//Reading dataset 11
R011: L     "SYS_DirectCtrlLCDB".PC.ObjectNo;
      L     #Par.ParObjectNo;
      <>I;
      JC    R101;
      AN    "SYS_DirectCtrlLCDB".PC.Hsk.FExamineFirst;
      AN    "SYS_DirectCtrlLCDB".PC.Hsk.FExamineNext;
      JC    R101;
// -- Start Reading with Dataset 11
      L     11;
      T     #DPData.NrRcvDataSet;
      L     253;	//First
      A     "SYS_DirectCtrlLCDB".PC.Hsk.FExamineFirst;
      JC    rLC9;
      L     254;	//Next
rLC9: T     #DPData.IdxRcvDataSet;
      JU    rcv0;
//<--[7.0]
//===============================
//Read Dataset 001 Index 1
R101: L     1;
      T     #DPData.NrRcvDataSet;
      L     1;
      T     #DPData.IdxRcvDataSet;
      A     #Par.HelpFlags.OutFaultResetDone;
      S     #Par.HelpFlags.OutFlagFaultResetDone;
      JU    rcv0;
//===============================
//Read Dataset 001 Index2
R201: L     1;
      T     #DPData.NrRcvDataSet;
      L     2;
      T     #DPData.IdxRcvDataSet;
      JU    rcv0;
//===============================
//Read Dataset 2
R002: L     2;
      T     #DPData.NrRcvDataSet;
      L     0;
      T     #DPData.IdxRcvDataSet;
      A     #Par.HelpFlags.OutFlagFaultResetDone;
      R     #Par.HelpFlags.OutFaultResetDone;
      R     #Par.HelpFlags.OutFlagFaultResetDone;
      S     #Par.HelpFlags.OutTestNewAlarm;
      JU    rcv0;
//===============================
//Read Dataset 3
R003: L     3;
      T     #DPData.NrRcvDataSet;
      L     0;
      T     #DPData.IdxRcvDataSet;
      JU    rcv0;
//===============================
rcv0: NOP   0;
      A     #Par.HelpFlags.OutComFaultRead;
      O     #Par.HelpFlags.OutComFaultSend;
      =     #OutComFault;
//-> IBS 2.12.06/Tho: [1.4] 
//   Delete actual values as long Profibus Fault
      JCN   res0;
      L     0;	//Lade NULL
      T     #tmpCnt;	// in ein temp. DW
      CALL  "SIEMENS_FILL" (
           BVAL                     := #tmpCnt,
           RET_VAL                  := #tmpRetVal,
           BLK                      := #Mill1.Act);	//Act.Mill1 auf Nullsetzen !!
      CALL  "SIEMENS_FILL" (
           BVAL                     := #tmpCnt,
           RET_VAL                  := #tmpRetVal,
           BLK                      := #Mill2.Act);	//Act. Mill2 auf Nullsetzen !!
      CALL  "SIEMENS_FILL" (
           BVAL                     := #tmpCnt,
           RET_VAL                  := #tmpRetVal,
           BLK                      := #Status);	//Status auf Nullsetzen !!
      CALL  "SIEMENS_FILL" (
           BVAL                     := #tmpCnt,
           RET_VAL                  := #tmpRetVal,
           BLK                      := #Command);	//Command auf Nullsetzen !!
      CALL  "SIEMENS_FILL" (
           BVAL                     := #tmpCnt,
           RET_VAL                  := #tmpRetVal,
           BLK                      := #OutpDFCO);	//OutpDFCO auf Nullsetzen !!
      CALL  "SIEMENS_FILL" (
           BVAL                     := #tmpCnt,
           RET_VAL                  := #tmpRetVal,
           BLK                      := #InpDFCO);	//InpDFCO auf Nullsetzen !!
res0: NOP   0;
//<-
NETWORK
TITLE = State Motor Mil1 1
      SET;
      R     #Mill1.Motor.StStopping;
      R     #Mill1.Motor.StStarting;
      R     #Mill1.Motor.StStopped;
      R     #Mill1.Motor.StBrake;
      R     #Mill1.Motor.StStopped;
      R     #Mill1.Motor.StStartedFwd;
      R     #Mill1.Motor.StStartedRev;
      R     #Mill1.Motor.StFault;
      L     #Mill1.Act.OutStatusMillMotor;
      JL    M1XX;	//Else
      JU    M1V0;
      JU    M1V1;
      JU    M1V2;
      JU    M1V3;
      JU    M1V4;
      JU    M1V5;
      JU    M1V6;
      JU    M1V7;
M1XX: JU    M1V6;
M1V0: L     0;
      JU    M1J9;
M1V1: S     #Mill1.Motor.StStopping;
      L     7;	// StCode.Stopping
      JU    M1J9;
M1V2: S     #Mill1.Motor.StBrake;
      L     7;	// StCode.Stopping
      JU    M1J9;
M1V3: S     #Mill1.Motor.StStopped;
      L     1;	// StCode.StStopped
      JU    M1J9;
M1V4: S     #Mill1.Motor.StStartedFwd;
      A     #Status.O82MotorFast1;
      L     4;	// StCode.StStartedFwdFast
      JC    M1J9;
      L     3;	// StCode.StStartedFwdSlow
      JU    M1J9;
M1V5: S     #Mill1.Motor.StStartedRev;
      A     #Status.O82MotorFast1;
      L     6;	// StCode.StStartedRevFast
      JC    M1J9;
      L     5;	// StCode.StStartedRevSlow
      JU    M1J9;
M1V6: S     #Mill1.Motor.StStarting;
      L     2;	// StCode.Starting
      JU    M1J9;
M1V7: S     #Mill1.Motor.StFault;
      L     32;	// StCode.Fault
M1J9: T     #Mill1.Motor_StCode;
NETWORK
TITLE = State Motor Mil1 2
      SET;
      R     #Mill2.Motor.StStopping;
      R     #Mill2.Motor.StStarting;
      R     #Mill2.Motor.StStopped;
      R     #Mill2.Motor.StBrake;
      R     #Mill2.Motor.StStopped;
      R     #Mill2.Motor.StStartedFwd;
      R     #Mill2.Motor.StStartedRev;
      R     #Mill2.Motor.StFault;
      L     #Mill2.Act.OutStatusMillMotor;
      JL    M2XX;	//Else
      JU    M2V0;
      JU    M2V1;
      JU    M2V2;
      JU    M2V3;
      JU    M2V4;
      JU    M2V5;
      JU    M2V6;
      JU    M2V7;
M2XX: JU    M2V7;	//Else
M2V0: L     0;
      JU    M2J9;
M2V1: S     #Mill2.Motor.StStopping;
      L     7;	// StCode.Stopping
      JU    M2J9;
M2V2: S     #Mill2.Motor.StBrake;
      L     7;	// StCode.Stopping
      JU    M2J9;
M2V3: S     #Mill2.Motor.StStopped;
      L     1;	//  StCode.StStopped
      JU    M2J9;
M2V4: S     #Mill2.Motor.StStartedFwd;
      A     #Status.O92MotorFast2;
      L     4;	// StCode.StStartedFwdFast
      JC    M2J9;
      L     3;	// StCode.StStartedFwdSlow
      JU    M2J9;
M2V5: S     #Mill2.Motor.StStartedRev;
      A     #Status.O92MotorFast2;
      L     6;	//  StCode.StStartedRevFast
      JC    M2J9;
      L     5;	//  StCode.StStartedRevFast
      JU    M2J9;
M2V6: S     #Mill2.Motor.StStarting;
      L     2;	// StCode.Starting
      JU    M2J9;
M2V7: S     #Mill2.Motor.StFault;
      L     32;	//  StCode.Fault
M2J9: T     #Mill2.Motor_StCode;
NETWORK
TITLE = State Flap Box
//[1.2] Tho: div. Korrekturen Sprungziele
//von LC: 
//1=Klappe nicht definiert
//2=Klappe Position Mühle 1
//3=Klappe in Mittelposition
//4=Klappe Position Mühle 2
      SET;
      R     #FlapBox.StMill1;
      R     #FlapBox.StMiddle;
      R     #FlapBox.StMill2;
      R     #FlapBox.StNoPosition;
      L     #Mill1.Act.OutStatusFlapBox;
      JL    FBXX;	//Else
      JU    FBV0;
      JU    FBV1;
      JU    FBV2;
      JU    FBV3;
      JU    FBV4;
FBXX: NOP   0;
FBV0: L     0;
      JU    FBJ9;
FBV1: SET;
      S     #FlapBox.StNoPosition;
      L     5;	// StCode.StNoPosition
      JU    FBJ9;
FBV2: SET;
      S     #FlapBox.StMill1;
      L     1;	// StCode.StMill1
      JU    FBJ9;
FBV3: SET;
      S     #FlapBox.StMiddle;
      L     6;	// StCode.StMiddle
      JU    FBJ9;
FBV4: S     #FlapBox.StMill2;
      L     3;	// StCode.StMill2
      JU    FBJ9;
FBJ9: T     #FlapBox_StCode;
NETWORK
TITLE = Status Addition Elements Mill 1
      NOP   0;
//===================================
//Vibration 
//===================================
      L     3;	//StCode=StTrue
      A     #InpDFCO.I60_VibrationDetector1;
      JC    SE1A;
      L     1;	//StCode=StFalse
SE1A: T     #Mill1.Vibration_StCode;
//===================================
//Automatic (1=Hand)
//===================================
      L     3;	//StCode=StTrue
      AN    #InpDFCO.I22_KeySwitchAuto1;	//[1.3]
      JC    SE1B;
      L     1;	//StCode=StFalse
SE1B: T     #Mill1.Automatic_StCode;
//===================================
//StandStill 
//===================================
      L     3;	//StCode=StTrue
      A     #InpDFCO.I24_StandStill1;
      JC    SE1C;
      L     1;	//StCode=StFalse
SE1C: T     #Mill1.StandStill_StCode;
//===================================
//ConnectingBlock 
//===================================
      L     3;	//StCode=StTrue
      A     #InpDFCO.I23_SwitchPanel1;
      JC    SE1D;
      L     1;	//StCode=StFalse
SE1D: T     #Mill1.SwitchPanel_StCode;
//===================================
//EmergencyStop 
//===================================
      L     3;	//StCode=StTrue
      A     #InpDFCO.I26_EmergencySwitch1;
      JC    SE1E;
      L     1;	//StCode=StFalse
SE1E: T     #Mill1.EmergencyStop_StCode;
//===================================
//HLCone 
//===================================
      L     3;	//StCode=StTrue
      AN    #InpDFCO.I27_HL_Cone1;
      JC    SE1F;
      L     1;	//StCode=StFalse
SE1F: T     #Mill1.HLCone_StCode;
NETWORK
TITLE = Status Addition Elements Mill 2
      NOP   0;
//===================================
//Vibration 
//===================================
      L     3;	//StCode=StTrue
      A     #InpDFCO.I61_VibrationDetector2;
      JC    SE2A;
      L     1;	//StCode=StFalse
SE2A: T     #Mill2.Vibration_StCode;
//===================================
//Automatic (1=Hand)
//===================================
      L     3;	//StCode=StTrue
      AN    #InpDFCO.I42_KeySwitchAuto2;	//[1.3]
      JC    SE2B;
      L     1;	//StCode=StFalse
SE2B: T     #Mill2.Automatic_StCode;
//===================================
//StandStill 
//===================================
      L     3;	//StCode=StTrue
      A     #InpDFCO.I44_StandStill2;
      JC    SE2C;
      L     1;	//StCode=StFalse
SE2C: T     #Mill2.StandStill_StCode;
//===================================
//ConnectingBlock 
//===================================
      L     3;	//StCode=StTrue
      A     #InpDFCO.I43_SwitchPanel2;
      JC    SE2D;
      L     1;	//StCode=StFalse
SE2D: T     #Mill2.SwitchPanel_StCode;
//===================================
//EmergencyStop 
//===================================
      L     3;	//StCode=StTrue
      A     #InpDFCO.I46_EmergencySwitch2;
      JC    SE2E;
      L     1;	//StCode=StFalse
SE2E: T     #Mill2.EmergencyStop_StCode;
//===================================
//HLCone 
//===================================
      L     3;	//StCode=StTrue
      AN    #InpDFCO.I47_HL_Cone2;
      JC    SE2F;
      L     1;	//StCode=StFalse
SE2F: T     #Mill2.HLCone_StCode;
NETWORK
TITLE = Status Addition Elements Mill 1 + 2
      NOP   0;
//===================================
//FeedRoll 
//===================================
      L     #OutActFeedRoll;	//[1.2]
      L     0;	//[1.2]
      >I;	//[1.2]
      L     3;	//StCode=StStartedFwd
      JC    SE3A;
      L     1;	//StCode=StFalse
SE3A: T     #FeedRoll_StCode;
//===================================
//LL_FeedHopper 
//===================================
      L     3;	//StCode=StTrue
      A     #InpDFCO.I00_LL_FeedHopper;
      JC    SE3B;
      L     1;	//StCode=StFalse
SE3B: T     #LL_FeedHopper_StCode;
//===================================
//HL_DFAV
//===================================
      L     3;	//StCode=StTrue
      AN    #InpDFCO.I01_HL_DFAV;	//[V1.2a] Tho: invertiert
      JC    SE3C;
      L     1;	//StCode=StFalse
SE3C: T     #HL_DFAV_StCode;
//===================================
//MagnetDoor
//===================================
      L     3;	//StCode=StTrue
      A     #InpDFCO.I03_MagnetDoorClosed;
      JC    SE3D;
      L     1;	//StCode=StFalse
SE3D: T     #MagnetDoor_StCode;
//===================================
//Fan
//===================================
      L     3;	//StCode=StStartedFwd
//[V1.2a] I83 meldet nicht, aber AckFanStart 
//      U     #InpDFCO.I83_AckFan
      A     #Command.AckFanStart;
      JC    SE3E;
      L     1;	//StCode=StFalse
SE3E: T     #Fan_StCode;
//===================================
//HeavyParticleFlap
//===================================
      L     3;	//StCode=StTrue
      A     #InpDFCO.I02_HeavyParticleFlap;
      JC    SE3F;
      L     1;	//StCode=StFalse
SE3F: T     #HeavyParticalFlap_StCode;
NETWORK
TITLE =  All State Init
      NOP   0;
//===Global Group Orders===
      A     "GCS7_Gr_OutManualOff";	//Gr.OutManualOff
      R     #InManual;
      A     #InManual;
      S     "GCS7_Gr_InManual";	//Gr.InManualMode
      A     "GCS7_Gr_OutFaultReset";	//Gr.OutOutFaultReset
      S     #CmdFaultReset;
//---Report is on---
      A     "GCS7_Gr_OutReportAll";	//Gr.OutReportAll
      O     #InReport;
      =     #tmpReport;
//---Local---
      A     #InLocal;
      AN    #InManual;
      =     #tmpLocal;
//--- fault
      A(;
      L     #Mill1.Act.OutAlarmNo;	//[2.1]
      L     0;	//[2.1]
      >I;	//[2.1]
      O(;	//[2.1]
      L     #Mill2.Act.OutAlarmNo;	//[2.1]
      L     0;	//[2.1]
      >I;	//[2.1]
      );	//[2.1]
      );	//[2.1]
      A     #Status.SumFault;
      O     #OutComFault;
      O     #Mill1.OutWrongValue;
      O     #Mill2.OutWrongValue;
      ON    #Status.RemoteControlDP;	//[6.2]
      AN    #tmpLocal;
      AN    #InHWStop;
      AN    #InDPFault;
      =     #tmpFault;
//---tmpStarted
      A     #Mill1.Motor.StStartedFwd;
      O     #Mill1.Motor.StStartedRev;
      ON    #Command.UsedMill1;
      A(;
      A     #Mill2.Motor.StStartedFwd;
      O     #Mill2.Motor.StStartedRev;
      ON    #Command.UsedMil12;
      );
      A(;
      O     #Command.UsedMill1;
      O     #Command.UsedMil12;
      );
      AN    #Par.ParDFCO_Only;
      O(;
      L     #OutActFeedRoll;
      L     0;
      >I;
      A     #Par.ParDFCO_Only;
      );
      =     #tmpStarted;
//--- tmpStopped
      A     #Mill1.Motor.StStopped;
      A     #Mill2.Motor.StStopped;
      AN    #Par.ParDFCO_Only;
      O(;
      L     #OutActFeedRoll;
      L     0;
      <=I;
      A     #Par.ParDFCO_Only;
      );
      =     #tmpStopped;
//----Loaded ------
      A     #Status.Loaded1;
      =     #Mill1.OutLoaded;
      A     #Status.Loaded2;
      =     #Mill2.OutLoaded;
NETWORK
TITLE = States
//===State machine===
      A     #StStopped;
      JC    S0;
      A     #StStarting;
      JC    S1;
      A     #StStarted;
      JC    S2;
      A     #StStopping;
      JC    S3;
      A     #StFault;
      JC    S4;
      S     #StStopped;	//Init
NETWORK
TITLE = StStopped
//Transition to StStopped
//Transition
xxS0: S     #StStopped;
      JU    LOGX;
//----------------------------------------------
//Logic
//Condition for StFault
S0:   A     #tmpFault;
      R     #StStopped;
      JC    xxS4;
//Condition for StStarting
      AN    #tmpStopped;
      R     #StStopped;
      JC    xxS1;
      JU    OUT;
NETWORK
TITLE =  STARTING
// Any Transition
//Transition
xxS1: S     #StStarting;
      JU    OUT;
//----------------------------------------------
//Logic
//Condition for StFault
S1:   A     #tmpFault;
      R     #StStarting;
      JC    xxS4;
//Condition for StStopping
      AN    #Mill1.InEnable;
      ON    #Mill1.InUsed;
      A(;
      AN    #Mill2.InEnable;
      ON    #Mill2.InUsed;
      );
      AN    #Par.ParDFCO_Only;
      O     #tmpStopped;
      R     #StStarting;
      JC    xxS3;
//-- Transition to Started --         
      A     #tmpStarted;
      R     #StStarting;
      JC    xxS2;
      JU    OUT;
NETWORK
TITLE = Started
//Transition
//----------------------------------------------
xxS2: SET;
      S     #StStarted;
      JU    LOGX;
//----------------------------------------------
//Condition for StFault
S2:   A     #tmpFault;
      R     #StStarted;
      JC    xxS4;
//Condition for StStarted
      A     #tmpStarted;
      JC    OUT;
//Condition for StStopping
      R     #StStarted;
      JC    xxS3;
      JU    OUT;
NETWORK
TITLE =  FAULT
//Condition for StStopped 
S4:   A     #Par.HelpFlags.OutTestNewAlarm;
      AN    #tmpFault;
      O;
      A     #InLocal;
      AN    #InManual;
      JC    S4S0;
      A     #Par.HelpFlags.OutTestNewAlarm;	//[2.3] Relog fault
      A     #tmpFault;	//[2.3]
      JC    xxS4;	//[2.3]
      JU    OUT;
//Transition to StStopped 
S4S0: S     #StStopped;
      R     #StFault;
      JU    LOG2;	//-->//Message ('fault cancelled')
NETWORK
TITLE =  StStopping
//Transition
//----------------------------------------------
xxS3: S     #StStopping;
      JU    OUT;
//----------------------------------------------
// Condition for fault
S3:   A     #tmpFault;
      R     #StStopping;
      JC    xxS4;
// Condition for Started
      A     #tmpStarted;
      R     #StStopping;
      JC    xxS2;
// Condition for stopped
      A     #tmpStopped;
      R     #StStopping;
      JC    xxS0;
      JU    OUT;
NETWORK
TITLE = LOG
////[5.0] Alarmnummer
xxS4: S     "GCS7_Gr_InFaultFlag";	//Gr.InFaultFlag
      S     #StFault;
//Horn On
      CALL  "SYS_Horn_Code" (
           FcCode                   := 1,
           ParObjectType            := 1040,
           ParObjectNo              := #Par.ParObjectNo,
           ParHornCode              := #Par.ParHornCode);
//Alarm Communication
      L     B#(1, 96);
      A     #OutComFault;
      JC    LOG;
//Alarm-Nr 1..80
      L     0;
      L     #Mill1.Act.OutAlarmNo;
      ==I;
      JC    LGM2;
      L     B#(1, 0);
      OW;
      JU    LOG;	//Alarms 1..80
//Alarm-Nr 1..80
LGM2: L     0;
      L     #Mill2.Act.OutAlarmNo;
      ==I;
      JC    LGM3;
      L     B#(1, 0);
      OW;
      JU    LOG;	//Alarms 1..80
//Fault Remote Control
LGM3: L     B#(1, 90);	// Message ('fault DP Mode')   //[6.2]
      AN    #Status.RemoteControlDP;	//[6.2]
      JC    LOG;	//[6.2]
//Wrong Value
      A     #Mill1.OutWrongValue;
      O     #Mill1.OutWrongValue;
      L     B#(1, 95);	// Message ('fault wrong value')
      JC    LOG;
//Collected Alarm
      L     B#(1, 99);	// Message ('fault collected alarm')
      JU    LOG;
//Fault Canceled
LOG2: L     B#(4, 0);	// Message ('fault Fault Canceled')
      JU    LOG;
//===============================================
//State Transition
LOGX: AN    #tmpReport;
      JC    OUT;
      A     #StStopped;
      L     B#(4, 91);	//Message ('Stopped')
      JC    LOG;
      A     #StStarted;
      L     B#(4, 92);	//Message ('Started')
      JC    LOG;
      JC    OUT;
LOG:  A     #Par.ParLogOff;	//---Set LOG Message
      JC    OUT;
      T     #tmpLOGvalue;
      L     W#16#FF;
      AW;
      T     #OutAlarmNoLog;
      CALL  "GCS7_LogConvert" (
           ObjectNo                 := #Par.ParObjectNo,
           MsgType                  := #Par.ParMsgType,
           ClassMsgTxt              := #tmpLOGvalue,
           OType                    := 1040);	//LOG Message Converter / Entry / Contains Class and TextNo
OUT:  NOP   0;
NETWORK
TITLE = Prepare Command ScreenChange
      L     #Mill1.Tar.InScreen;
      L     #Mill1.OutScreenAct;
      <>I;
      =     #Mill1.OutScreenChangeReq;
      A     #Mill1.OutScreenChangeReq;
      =     #Command.ReqScreenChange1;
//------------------------------------
      L     #Mill2.Tar.InScreen;
      L     #Mill2.OutScreenAct;
      <>I;
      =     #Mill2.OutScreenChangeReq;
      A     #Mill2.OutScreenChangeReq;
      =     #Command.ReqScreenChange2;
//------------------------------------
//Screen change done Mill 1
      A     #Command.ReqScreenChange1;
      A     #Status.AckScreenChange1;
      JCN   SCS2;
      L     #Mill1.Tar.InScreen;
      T     #Mill1.OutScreenAct;
SCS2: NOP   0;
//------------------------------------
//Screen change done Mill 2 
      A     #Command.ReqScreenChange2;
      A     #Status.AckScreenChange2;
      JCN   SCS3;
      L     #Mill2.Tar.InScreen;
      T     #Mill2.OutScreenAct;
SCS3: NOP   0;
NETWORK
TITLE = Timeout time Mill 1
      A     #Mill1.Motor.StStopped;
      O     #Mill1.Motor.StFault;
      A     #Command.EnableMill1;
      AN    #Par.ParDFCO_Only;	// [2.3]
      JC    T1J1;
      L     #Par.ParTimeOutStart;
      T     #Par.OutTimeOutStart1;
      JU    T1J2;
T1J1: L     0;
      L     #Par.OutTimeOutStart1;
      >=I;
      ON    "GCS7_Gr_OutTick200ms";
      JC    T1J3;
      +     -2;
      T     #Par.OutTimeOutStart1;
T1J3: L     0;
      <=I;
      R     #Command.EnableMill1;
T1J2: NOP   0;
NETWORK
TITLE = Timeout time Mill 2
      A     #Mill2.Motor.StStopped;	//[1.2]
      O     #Mill2.Motor.StFault;
      A     #Command.EnableMill2;
      AN    #Par.ParDFCO_Only;	// [2.3]
      JC    T2J1;
      L     #Par.ParTimeOutStart;
      T     #Par.OutTimeOutStart2;
      JU    T2J2;
T2J1: L     0;
      L     #Par.OutTimeOutStart2;
      >=I;
      ON    "GCS7_Gr_OutTick200ms";
      JC    T2J3;
      +     -2;
      T     #Par.OutTimeOutStart2;
T2J3: L     0;
      <=I;
      R     #Command.EnableMill2;
T2J2: NOP   0;
NETWORK
TITLE = Prepare Command for MEAF
      NOP   0;
//==============================
      A     #Status.AcceptNewSendData;
      A     #Command.ResetAlarm;
      R     #Command.ResetAlarm;
      S     #Par.HelpFlags.OutFaultResetDone;
      AN    #Status.AcceptNewSendData;
      A     #CmdFaultReset;
      R     #CmdFaultReset;
      S     #Command.ResetAlarm;
//==============================
//Mill 1+2
//==============================
      A     #InHeavyFractionOpen;
      =     #Command.HeavyFractionOpen;
      A     #InManual;
      JC    CDJ1;
      A     #InReqStartRev;
      =     #Command.ReqStartRev;
      A     #InReqStartFwd;
      =     #Command.ReqStartFwd;
      A     #Mill1.InFast;
      =     #Command.MotorMill1Fast;
      A     #Mill2.InFast;
      =     #Command.MotorMill2Fast;
//==============================
//Mill 1
//==============================
CDJ1: A     #CmdNext;
      A     #Mill1.InEnable;
      AN    #InManual;
      O     #Mill1.CmdOn;
      S     #Command.EnableMill1;
      AN    #Mill1.InEnable;
      O     #Command.BrakeMill1;
      ON    #Mill1.InUsed;
      O     #tmpLocal;
      AN    #InManual;
      O     #Mill1.CmdOff;
      O     #Mill1.CmdBrake;
      R     #Command.EnableMill1;
//------------------------------
      A     #Mill1.InUsed;
      AN    #InManual;
      O;
      A     #InManual;
      A     #Command.EnableMill1;
      =     #Command.UsedMill1;
//------------------------------
      A     #Mill1.InEnableFeed;
      AN    #InManual;
      O     #Mill1.CmdFeedOn;
      S     #Command.EnableFeedMill1;
      AN    #Mill1.InEnableFeed;
      AN    #InManual;
      O     #Mill1.CmdFeedOff;
      ON    #Command.EnableMill1;
      R     #Command.EnableFeedMill1;
//------------------------------
      A     #Mill1.InBrake;
      O     #Mill1.OutScreenChangeReq;
      AN    #InManual;
      O     #Mill1.CmdBrake;
      S     #Command.BrakeMill1;
      AN    #Mill1.InBrake;
      AN    #Mill1.OutScreenChangeReq;
      AN    #InManual;
      O     #Mill1.Motor.StStopped;
      R     #Command.BrakeMill1;
//==============================
//Mill 2
//==============================
      A     #CmdNext;
      A     #Mill2.InEnable;
      AN    #InManual;
      O     #Mill2.CmdOn;
      S     #Command.EnableMill2;
      AN    #Mill2.InEnable;
      ON    #Mill2.InUsed;
      O     #tmpLocal;
      O     #Command.BrakeMill2;
      AN    #InManual;
      O     #Mill2.CmdOff;
      O     #Mill2.CmdBrake;
      R     #Command.EnableMill2;
//------------------------------
      A     #Mill2.InUsed;
      AN    #InManual;
      O;
      A     #InManual;
      A     #Command.EnableMill2;
      =     #Command.UsedMil12;
//------------------------------
      A     #Mill2.InEnableFeed;
      AN    #InManual;
      O     #Mill2.CmdFeedOn;
      S     #Command.EnableFeedMill2;
      AN    #Mill2.InEnableFeed;
      AN    #InManual;
      O     #Mill2.CmdFeedOff;
      ON    #Command.EnableMill2;
      R     #Command.EnableFeedMill2;
//------------------------------
      A     #Mill2.InBrake;
      O     #Mill2.OutScreenChangeReq;
      AN    #InManual;
      O     #Mill2.CmdBrake;
      S     #Command.BrakeMill2;
      AN    #Mill2.InBrake;
      AN    #Mill2.OutScreenChangeReq;
      AN    #InManual;
      O     #Mill2.Motor.StStopped;
      R     #Command.BrakeMill2;
//===============================
//AckStartRequest
//===============================
      A     #Status.ReqStartRequest;
      AN    "GCS7_Gr_InHeavyStartup";
      S     #Command.AckStartRequest;
      =     #tmpBool;	//[2.2]
      A     #tmpBool;	//[2.2]
      AN    #Par.ParDFCO_Only;	//[2.2]
      S     "GCS7_Gr_InHeavyStartup";
      AN    #Status.ReqStartRequest;
      O     #OutComFault;
      A     #Command.AckStartRequest;
      R     #Command.AckStartRequest;
      =     #tmpBool;	//[2.2]
      A     #tmpBool;	//[2.2]
      AN    #Par.ParDFCO_Only;	//[2.2]
      R     "GCS7_Gr_InHeavyStartup";
//==============================
      A     #Status.NewDataReady;
      =     #Command.AcceptNewDataReady;
//==============================
      SET;
      =     #Command.CommandReady;
//==============================
      A     #Status.NewRcvData;
      =     #Command.AcceptNewRcvData;
//==============================
      AN    #Status.AcceptNewSendData;
      =     #Command.NewSendData;
NETWORK
TITLE = Write Digital Outputs/ Read Digital Inputs
      A     #Mill1.InpFanStart;
      =     #Command.AckFanStart;
      A     #Status.O81MotorFwd1;
      AN    #OutComFault;
      =     #Mill1.OutpMotorFwd;
      A     #Status.O82MotorFast1;
      AN    #OutComFault;
      =     #Mill1.OutpMotorFast;
      A     #Status.O83MotorRev1;
      AN    #OutComFault;
      =     #Mill1.OutpMotorRev;
      A     #Status.O84Brake1;
      AN    #OutComFault;
      =     #Mill1.OutpBrake;
      A     #Status.O85FanStart;
      AN    #OutComFault;
      =     #Mill1.OutpFanStart;
      A     #Status.O91MotorFwd2;
      AN    #OutComFault;
      =     #Mill2.OutpMotorFwd;
      A     #Status.O92MotorFast2;
      AN    #OutComFault;
      =     #Mill2.OutpMotorFast;
      A     #Status.O93MotorRev2;
      AN    #OutComFault;
      =     #Mill2.OutpMotorRev;
      A     #Status.O94Brake2;
      AN    #OutComFault;
      =     #Mill2.OutpBrake;
NETWORK
TITLE = (Profibus) Send Data
//------------------------------------------------
//Test Send Dataset 128 Index 1 done
      L     #DPData.NrSndDataSet;
      L     128;
      <>I;
      O(;
      L     #DPData.IdxSndDataSet;
      L     1;
      <>I;
      );
      JC    s228;
      A     #Status.WrongValue;
      =     #Mill1.OutWrongValue;
      JU    S228;	//-->Send 128 Index 2
//------------------------------------------------
//Test Send Dataset 128 Index 2 done
s228: L     #DPData.NrSndDataSet;
      L     128;
      <>I;
      O(;
      L     #DPData.IdxSndDataSet;
      L     2;
      <>I;
      );
      JC    S128;
      A     #Status.WrongValue;
      =     #Mill2.OutWrongValue;
      JU    S128;	//-->Send 128 Index 1
//==================================================
//Send Dataset 128 Index 1
S128: L     128;
      T     #DPData.NrSndDataSet;
      L     1;
      T     #DPData.IdxSndDataSet;
      CALL  "SIEMENS_BLKMOV" (
           SRCBLK                   := #Mill1.Tar,
           RET_VAL                  := #tmpReturn,
           DSTBLK                   := #DPData.Data);
      JU    Snd;
//======================================================
//Send Dataset 128 Index 2
S228: L     128;
      T     #DPData.NrSndDataSet;
      L     2;
      T     #DPData.IdxSndDataSet;
      CALL  "SIEMENS_BLKMOV" (
           SRCBLK                   := #Mill2.Tar,
           RET_VAL                  := #tmpReturn,
           DSTBLK                   := #DPData.Data);
      JU    Snd;
//======================================================
//Senden DP
Snd:  CALL  "SIEMENS_BLKMOV" (
           SRCBLK                   := #Command,
           RET_VAL                  := #tmpReturn,
           DSTBLK                   := #DPData.StatusCommand);
      A     #InSimulation;
      JC    sSim;
      CALL  "SIEMENS_DPWR_DAT" (
           LADDR                    := #tmpAddr,
           RECORD                   := #DPData,
           RET_VAL                  := #tmpReturn);
      L     #tmpReturn;
      L     0;
      <>I;
      =     #Par.HelpFlags.OutComFaultSend;
      JU    sEnd;
//write to Simulation
sSim: R     #Par.HelpFlags.OutComFaultSend;
      A     "GCS7_Gr_SimDPtoImage";
      L     P#Q 0.0;
      JC    rDB2;
      OPN   "TEST_IOSimuliOutput";
      L     P#DBX 0.0;
rDB2: L     #Par.ParIOByteNo;
      SLD   3;
      +D;
      LAR1;
      L     #DPData.StatusCommand;
      T     D [AR1,P#0.0];
      L     #DPData.NrSndDataSet;
      T     B [AR1,P#4.0];
      L     #DPData.IdxSndDataSet;
      T     B [AR1,P#5.0];
      L     #DPData.NrRcvDataSet;
      T     B [AR1,P#6.0];
      L     #DPData.IdxRcvDataSet;
      T     B [AR1,P#7.0];
      L     #DPData.Data[1];
      T     D [AR1,P#8.0];
      L     #DPData.Data[2];
      T     D [AR1,P#12.0];
      L     #DPData.Data[3];
      T     D [AR1,P#16.0];
      L     #DPData.Data[4];
      T     D [AR1,P#20.0];
sEnd: NOP   0;
      NOP   0;
NETWORK
TITLE = Global End
      SET;	//---Clear commands
      R     #CmdNext;
      R     #Par.HelpFlags.OutTestNewAlarm;
      R     #Mill1.CmdOff;
      R     #Mill1.CmdOn;
      R     #Mill1.CmdFeedOff;
      R     #Mill1.CmdFeedOn;
      R     #Mill1.CmdBrake;
      R     #Mill2.CmdOff;
      R     #Mill2.CmdOn;
      R     #Mill2.CmdFeedOff;
      R     #Mill2.CmdFeedOn;
      R     #Mill2.CmdBrake;
//--Output for group 
      A     #InDPFault;
      AN    #tmpLocal;
      S     "GCS7_Gr_InDPFault";
      A     #InHWStop;
      AN    #tmpLocal;
      S     "GCS7_Gr_InHWStop";
      A     #StFault;
      S     "GCS7_Gr_InFault";	// Gr.InFault
NETWORK
TITLE = State Code
// State                 StCode
// -----------------------------
// StFault                 32
// StStopped                1
// StStarting               2
// StStarted.Wait           3
// StStarted.Feeding        4
// StStopping               7
// StWarning                8
      A     #StStopped;
      L     1;	//Code=StStopped
      JC    Code;
      L     #OutActFeedRoll;
      L     0;
      >I;
      A     #StStarted;
      L     4;	//Code= StStarted.Feeding
      JC    Code;
      A     #StStarted;
      L     3;	//Code=StStarted.Wait
      JC    Code;
      A     #StStarting;
      L     2;	//Code=StStarting
      JC    Code;
      A     #StStopping;
      L     7;	//Code=StStopping 
      JC    Code;
      L     32;	//Code=StFault 
Code: T     #StCode;	// Save state code
NETWORK
TITLE = Timer/Counter Mill 1
      NOP   0;
//-----------------------------------
      AN    #Mill1.Motor.StStartedFwd;
      ON    "GCS7_Gr_OutTick1s";
      JC    T1RV;
      L     #Mill1.OutTimeStartedFwd;
      +     L#1;
      T     #Mill1.OutTimeStartedFwd;
//-----------------------------------
T1RV: AN    #Mill1.Motor.StStartedRev;
      ON    "GCS7_Gr_OutTick1s";
      JC    T1CS;
      L     #Mill1.OutTimeStartedRev;
      +     L#1;
      T     #Mill1.OutTimeStartedRev;
//-----------------------------------
T1CS: A     #Mill1.Motor.StStartedFwd;
      O     #Mill1.Motor.StStartedRev;
      FP    #Mill1.VarEdgeStarted;
      JCN   T1CF;
      L     #Mill1.OutCntStartup;
      +     L#1;
      T     #Mill1.OutCntStartup;
//-----------------------------------
T1CF: L     #Mill1.Act.OutAlarmNo;
      L     0;
      <>I;
      A     #StFault;
      FP    #Mill1.VarEdgeFault;
      JCN   T1J9;
      L     #Mill1.OutCntFault;
      +     L#1;
      T     #Mill1.OutCntFault;
T1J9: NOP   0;
NETWORK
TITLE = Timer/Counter Mill 2
      NOP   0;
//-----------------------------------
      AN    #Mill2.Motor.StStartedFwd;
      ON    "GCS7_Gr_OutTick1s";
      JC    T2RV;
      L     #Mill2.OutTimeStartedFwd;
      +     L#1;
      T     #Mill2.OutTimeStartedFwd;
//-----------------------------------
T2RV: AN    #Mill2.Motor.StStartedRev;
      ON    "GCS7_Gr_OutTick1s";
      JC    T2CS;
      L     #Mill2.OutTimeStartedRev;
      +     L#1;
      T     #Mill2.OutTimeStartedRev;
//-----------------------------------
T2CS: A     #Mill2.Motor.StStartedFwd;
      O     #Mill2.Motor.StStartedRev;
      FP    #Mill2.VarEdgeStarted;
      JCN   T2CF;
      L     #Mill2.OutCntStartup;
      +     L#1;
      T     #Mill2.OutCntStartup;
//-----------------------------------
T2CF: L     #Mill2.Act.OutAlarmNo;
      L     0;
      <>I;
      A     #StFault;
      FP    #Mill2.VarEdgeFault;
      JCN   T2J9;
      L     #Mill2.OutCntFault;
      +     L#1;
      T     #Mill2.OutCntFault;
T2J9: NOP   0;
END_FUNCTION_BLOCK

